RoboDK station: Stitching with sticher.rdk

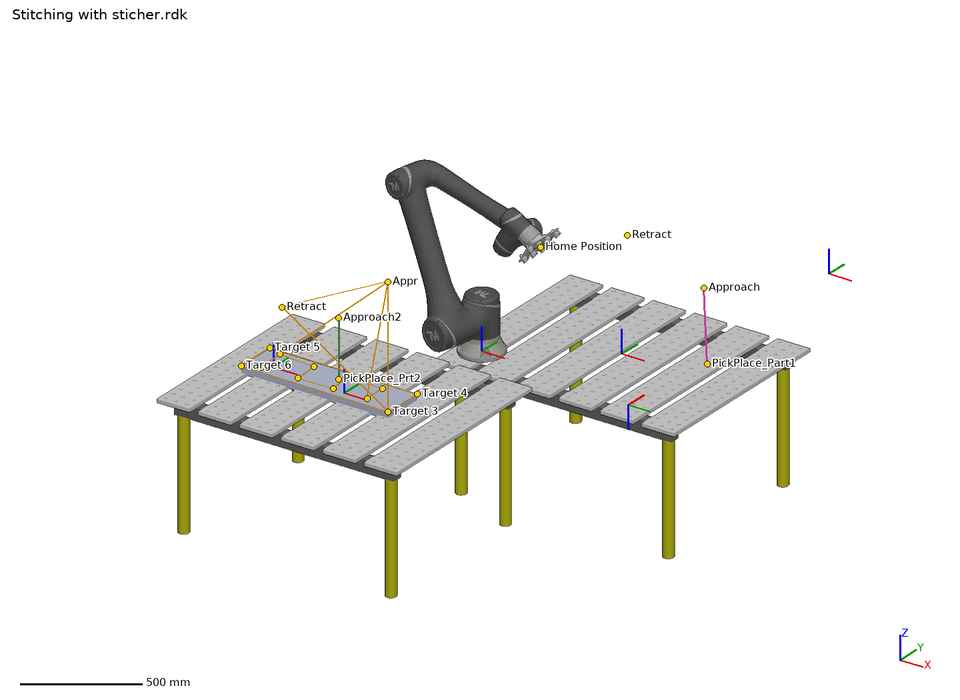
[picture v0: the station drawn from its stored meshes, robots at their saved joint values, targets as dots, program paths as lines]
Station Stitching with sticher (saved by RoboDK 5.1.0). Poses are relative to the parent item; angles as X-Y-Z fixed-axis rotations.
Station parameters (name, value as stored): OPC-UA, opc.tcp://localhost:4840
  - frame Omron TM12X Base at (-746.68, 425.35, 0) mm
    - robot Omron TM12X: 6 axes, payload 12 kg, reach 1300 mm, repeatability 0.1 mm, weight 33.3 kg
        modified DH rows (alpha deg, a mm, theta deg, d mm): 0, 0, 0, 165.2; 90, 0, 90, 0; 0, 636.1, 0, 0; 0, 557.9, -90, 156.3; -90, 0, 0, 106; 90, 0, 180, 113.15
        joint limits [-270, -180, -166, -180, -180, -270] to [270, 180, 166, 180, 180, 270]; home [0, 0, 90, 0, 90, 0]; saved at [-10.231, -22.802, 121.949, -69.746, 97.894, -185.07]
      - tool GripperA, TCP at (0, 0, 30) mm, rotated rx 0 ry 0 rz 90 deg, size 209.9 x 42 x 100 mm
  - frame Frame 2 at (-849.61, -404.11, 112.6) mm
    - target Home Position (Cartesian target) at (550.89, 609.76, 573.04) mm, rotated rx -178.84 ry 60.9 rz -179.86 deg; joints [-18.502, -38.59, 118.247, -49.418, 105.073, -99.264] of Omron TM12X
    - target Retract (Cartesian target) at (930.89, 679.76, 703.04) mm, rotated rx -173.84 ry 45.9 rz -174.86 deg; joints [2.137, -2.643, 73.991, -27.43, 86, -92.092] of Omron TM12X
    - target Approach (Cartesian target) at (924.81, 1233.71, 243.56) mm, rotated rx 179.4 ry 2.27 rz -178.66 deg; joints [36.144, 26.738, 88.534, -27.482, 89.197, -145.226] of Omron TM12X
    - target PickPlace_Part1 (Cartesian target) at (940.37, 1235.87, -99.57) mm, rotated rx -179.05 ry -0.07 rz -178.55 deg; joints [35.67, 47.381, 94.458, -51.245, 89.251, -145.772] of Omron TM12X
    - object Table at (0, 0, 0) mm, size 1193.8 x 965.2 x 609.6 mm, geometry from welding_table.sld
  - frame Object at (-329.47, 825.84, -55.54) mm
    - object Table at (0, 0, 0) mm, size 1193.8 x 965.2 x 609.6 mm, geometry from welding_table.sld
  - frame Pick at (-14.83, 419.35, -35.5) mm, rotated rx 179.89 ry 0 rz 89.08 deg
  - frame Drop at (-1209.15, -394.59, 123.51) mm
    - target Approach2 (Cartesian target) at (319.83, 8.55, 311.87) mm, rotated rx -178.81 ry -0.1 rz 92.19 deg; joints [-88.823, 16.471, 94.157, -20.547, 88.807, -181.01] of Omron TM12X
    - target PickPlace_Prt2 (Cartesian target) at (319.83, 8.55, 31.87) mm, rotated rx -178.81 ry -0.1 rz 92.19 deg; joints [-88.823, 30.903, 106.753, -47.575, 88.807, -181.01] of Omron TM12X
    - object 197143A at (-94.1, 108.82, -14.88) mm, rotated rx 179.92 ry 0.24 rz -0.18 deg, size 734 x 204 x 35 mm, geometry from 197143A.IGS
  - program ReplaceObjects (1 instructions, listed below)
  - program PickPart1 (6 instructions, listed below)
  - program PlacePart2 (6 instructions, listed below)
  - program PickPart2 (6 instructions, listed below)
  - program PlacePart1 (6 instructions, listed below)
  - program MainProgram (4 instructions, listed below)
  - frame Frame 7 at (0, 1825.84, 0) mm
    - target Appr (Cartesian target) at (-569.76, -2317.87, 730.86) mm, rotated rx -179.96 ry -0.25 rz -170 deg; joints [36.138, -4.221, 91.35, -32.89, 73.964, -69.08]
    - target Retract (Cartesian target) at (-789.76, -2757.87, 730.86) mm, rotated rx -179.96 ry -0.25 rz -170 deg; joints [2.404, -12.401, 102.683, -90.029, 97.595, -90.074]
    - target Target 3 (Cartesian target) at (-569.76, -2317.87, 140.86) mm, rotated rx -179.96 ry -0.25 rz -170 deg; joints [38.37, 26.575, 116.834, -108.562, 66.075, -74.281]
    - target Target 4 (Cartesian target) at (-569.12, -2113.87, 140.56) mm, rotated rx -179.96 ry -0.25 rz -170 deg; joints [49.798, 32.826, 104.437, -98.692, 56.897, -66.514]
    - target Target 5 (Cartesian target) at (-1303.11, -2111.56, 143.63) mm, rotated rx -179.96 ry -0.25 rz -170 deg; joints [119.416, -1.405, 133.583, -13.655, 36.472, 34.003]
    - target Target 6 (Cartesian target) at (-1303.75, -2315.56, 143.93) mm, rotated rx -179.96 ry -0.25 rz -170 deg; joints [138.762, -25.638, 146.558, 14.727, 48.34, 56.934]
    - target Target 7 (Cartesian target) at (-569.76, -2317.87, 140.86) mm, rotated rx -179.96 ry -0.25 rz -170 deg; joints [38.37, 24.049, 96.784, 94.013, -66.075, 105.719]
    - target Appr (Cartesian target) at (-569.76, -2317.87, 730.86) mm, rotated rx -179.96 ry -0.25 rz -170 deg; joints [36.138, -4.221, 91.35, -32.89, 73.964, -69.08]
    - target Target 9 (Cartesian target) at (-1230.22, -2278.33, 143.57) mm, rotated rx -179.96 ry -0.25 rz -170 deg; joints [122.87, -22.758, 147.645, -2.462, 38.225, 38.912]
    - target Target 10 (Cartesian target) at (-1236.06, -2136.84, 143.38) mm, rotated rx -179.96 ry -0.25 rz -170 deg; joints [113.503, -4.258, 138.046, -22.882, 33.993, 24.688]
    - target Target 11 (Cartesian target) at (-1056.31, -2149.37, 142.65) mm, rotated rx -179.96 ry -0.25 rz -170 deg; joints [91.788, 2.576, 141.142, -66.806, 32.426, -15.447]
    - target Target 12 (Cartesian target) at (-1047.71, -2275.5, 142.8) mm, rotated rx -179.96 ry -0.25 rz -170 deg; joints [90.995, -9.282, 152.029, -67.043, 32.614, -16.88]
    - target Target 13 (Cartesian target) at (-877.24, -2268.97, 142.08) mm, rotated rx -179.96 ry -0.25 rz -170 deg; joints [66.553, 9.069, 142.341, -103.375, 44.621, -51.687]
    - target Target 14 (Cartesian target) at (-893.9, -2153.07, 141.98) mm, rotated rx -179.96 ry -0.25 rz -170 deg; joints [73.078, 13.564, 134.273, -94.287, 40.49, -44.211]
    - target Target 15 (Cartesian target) at (-712.79, -2153.19, 141.22) mm, rotated rx -179.96 ry -0.25 rz -170 deg; joints [57.117, 23.688, 120.597, -102.284, 51.309, -60.673]
    - target Target 16 (Cartesian target) at (-711.23, -2264.87, 141.38) mm, rotated rx -179.96 ry -0.25 rz -170 deg; joints [50.89, 19.834, 127.999, -108.808, 56.046, -65.693]
    - target Appr (Cartesian target) at (-569.76, -2317.87, 730.86) mm, rotated rx -179.96 ry -0.25 rz -170 deg; joints [36.138, -4.221, 91.35, -32.89, 73.964, -69.08]
  - frame Frame 8 at (0, 2825.84, 0) mm
  - program Main Stich (19 instructions, listed below)
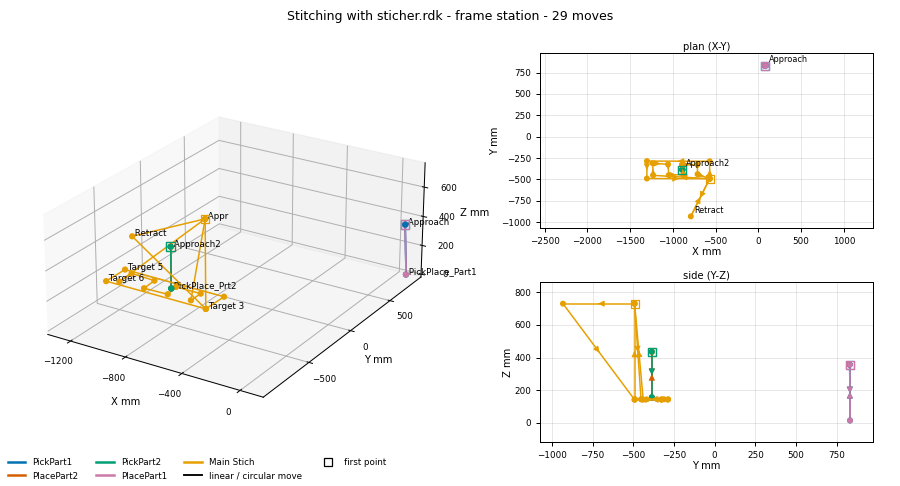
[picture p0: tool path of Stitching with sticher.rdk in frame station, 29 of 29 moves have a stored position in this frame; points joined in program order, loops and branches not executed]

--- program ReplaceObjects (robot Omron TM12X) ---
  Replace objects

--- program PickPart1 (robot Omron TM12X) ---
  Set Ref.: Frame 2
  Set Tool: GripperA
  MoveJ (Approach)
  MoveL (PickPlace_Part1)
  Attach to GripperA
  MoveL (Approach)

--- program PlacePart2 (robot Omron TM12X) ---
  Set Ref.: Drop
  Set Tool: GripperA
  MoveJ (Approach2)
  MoveL (PickPlace_Prt2)
  Detach from GripperA
  MoveL (Approach2)

--- program PickPart2 (robot Omron TM12X) ---
  Set Ref.: Drop
  Set Tool: GripperA
  MoveJ (Approach2)
  MoveL (PickPlace_Prt2)
  Attach to GripperA
  MoveL (PickPlace_Prt2)

--- program PlacePart1 (robot Omron TM12X) ---
  Set Ref.: Frame 2
  Set Tool: GripperA
  MoveJ (Approach)
  MoveL (PickPlace_Part1)
  Detach from GripperA
  MoveL (Approach)

--- program MainProgram (robot Omron TM12X) ---
  Call PickPart1
  Call PlacePart2
  Call PickPart2
  Call PlacePart1

--- program Main Stich ---
  Set Ref.: Frame 7
  Set Tool: Spindle at (186.14, 0, 258.61) mm, rotated rx 0 ry 58.76 rz 0 deg
  MoveJ (Appr)
  MoveL (Retract)
  MoveL (Target 3)
  MoveL (Target 4)
  MoveL (Target 5)
  MoveL (Target 6)
  MoveL (Target 7)
  MoveL (Appr)
  MoveL (Target 9)
  MoveL (Target 10)
  MoveL (Target 11)
  MoveL (Target 12)
  MoveL (Target 13)
  MoveL (Target 14)
  MoveL (Target 15)
  MoveL (Target 16)
  MoveL (Appr)
